// TIA Portal project "DT101" (V15.1)

(* hardware
DEVICE "S7-1200 station_1"  S7-1200 Station
   slot 0: "Rack_0"  S7-1200 Rack  Rack  V1.0
   slot 1: "PLC_1"  CPU 1214C AC/DC/Rly  6ES7 214-1BG40-0XB0  V4.2
      slot 3: "AQ 1x12BIT_1"  AQ1 signal board  6ES7 232-4HA30-0XB0  V1.0
   slot 101: "CM 1241 (RS485)_1"  CM 1241 (RS485)  6ES7 241-1CH30-0XB0  V1.0
DEVICE "GSD device_1"  GSD.Device.PN
   slot 0: "DTE101-PN"  DTE101-PN  DTE101  V1.1
      slot 0: "DTE101-PN"  DTE101-PN
      slot 1: "PROFINET-IO"  PROFINET-IO
         slot 1: "PORT 1"  PORT 1
         slot 2: "PORT 2"  PORT 2
   slot 0: "Rack"  Rack  V1.0
   slot 1: "INACTIVE_1"  INACTIVE  Output deactived
      slot 0: "INACTIVE"  INACTIVE
   slot 2: "RWH_RW_1"  RWH_RW  Read/write head
      slot 0: "RWH_RW"  RWH_RW
   slot 3: "INACTIVE_3"  INACTIVE  Output deactived
      slot 0: "INACTIVE"  INACTIVE
   slot 4: "INACTIVE_4"  INACTIVE  Output deactived
      slot 0: "INACTIVE"  INACTIVE
*)

// ===== PLC "PLC_1"  CPU 1214C AC/DC/Rly =====

ORGANIZATION_BLOCK "Main"   // OB1, LAD, ProgramCycle
TITLE = "Main Program Sweep (Cycle)"
{ S7_Optimized_Access := 'TRUE' }
VERSION : 0.1
   VAR_INPUT
      Initial_Call : Bool;   // Initial call of this OB
      Remanence : Bool;   // =True, if remanent data are available
   END_VAR
BEGIN
END_ORGANIZATION_BLOCK